NETWORK
TITLE = 1109 - MCC10.3_I811_MA3508 - Zone 1 Burner Fan - Motor

       CALL #"MCC10.3_I811_MA3508"
       (
         CM_No       := 1109 ,
         Unit       :=  ,
         Type       :=  ,
         Tab       := 28 ,
         SubTab       := 3 ,
         Safety       :=  ,
         Disconnect       := LCP131_I811_FN3508_DI_Flt ,
         Protect       := MCC10_I811_FC3508_DI_Flt ,
         RotationFB       :=  ,
         P2002_Current       :=  ,
         P2003_Torque       :=  ,
         P2001_RefVolt       := 460 ,
         EU_Ratio       :=  ,
         Gear_Ratio       :=  ,
         DeAct_Standstill       := T#30s ,
         ID_Free_telegram       :=  ,
         AmpRated       := 3,6 ,
         TorqueRated       :=  ,
         kWRated       := 1.5 ,
         SC_Local       := SL_28_S1 ,
         CM_FRQ        := "dbPlcHmiFRQ".FRQ[1109] ,
       );

NETWORK
TITLE = 1110 - MCC10.3_I521_MA3512 - Zone 2 Disc Filter Cleaning Fan - Motor

       CALL #"MCC10.3_I521_MA3512"
       (
         CM_No       := 1110 ,
         Unit       :=  ,
         Type       :=  ,
         Tab       := 28 ,
         SubTab       := 4 ,
         Safety       :=  ,
         Disconnect       := LCP131_I521_FN3512_DI_Flt ,
         Protect       := MCC10_I521_FC3512_DI_Flt ,
         RotationFB       :=  ,
         P2002_Current       :=  ,
         P2003_Torque       :=  ,
         P2001_RefVolt       := 460 ,
         EU_Ratio       :=  ,
         Gear_Ratio       :=  ,
         DeAct_Standstill       := T#30s ,
         ID_Free_telegram       :=  ,
         AmpRated       := 11 ,
         TorqueRated       :=  ,
         kWRated       := 7.5 ,
         SC_Local       := SL_28_S1 ,
         CM_FRQ        := "dbPlcHmiFRQ".FRQ[1110] ,
       );

NETWORK
TITLE = 1111 - MCC10.2_I621_MA3520 - Zone 2 Circulation Fan  - Motor

       CALL #"MCC10.2_I621_MA3520"
       (
         CM_No       := 1111 ,
         Unit       :=  ,
         Type       :=  ,
         Tab       := 28 ,
         SubTab       := 4 ,
         Safety       :=  ,
         Disconnect       := LCP102_I621_FN3520_DI_Flt ,
         Protect       := MCC10_I621_FC3520_DI_Flt ,
         RotationFB       :=  ,
         P2002_Current       :=  ,
         P2003_Torque       :=  ,
         P2001_RefVolt       := 460 ,
         EU_Ratio       :=  ,
         Gear_Ratio       :=  ,
         DeAct_Standstill       := T#30s ,
         ID_Free_telegram       :=  ,
         AmpRated       := 115 ,
         TorqueRated       :=  ,
         kWRated       := 7.5 ,
         SC_Local       := SL_28_S1 ,
         CM_FRQ        := "dbPlcHmiFRQ".FRQ[1111] ,
       );

NETWORK
TITLE = 1112 - MCC10.3_K911_MA3521 - Dryer 2 Sealing Fan  - Motor

       CALL #"MCC10.3_K911_MA3521"
       (
         CM_No       := 1112 ,
         Unit       :=  ,
         Type       :=  ,
         Tab       := 28 ,
         SubTab       := 1 ,
         Safety       :=  ,
         Disconnect       := LCP131_K911_FN3521_DI_Flt ,
         Protect       := MCC10_K911_FC3521_DI_Flt ,
         RotationFB       :=  ,
         P2002_Current       :=  ,
         P2003_Torque       :=  ,
         P2001_RefVolt       := 460 ,
         EU_Ratio       :=  ,
         Gear_Ratio       :=  ,
         DeAct_Standstill       := T#30s ,
         ID_Free_telegram       :=  ,
         AmpRated       := 5,8 ,
         TorqueRated       :=  ,
         kWRated       := 5.5 ,
         SC_Local       := SL_28_S2 ,
         CM_FRQ        := "dbPlcHmiFRQ".FRQ[1112] ,
       );

NETWORK
TITLE = 1113 - MCC10.3_K511_MA3522 - Zone 3 Disc Filter Cleaning Fan - Motor

       CALL #"MCC10.3_K511_MA3522"
       (
         CM_No       := 1113 ,
         Unit       :=  ,
         Type       :=  ,
         Tab       := 28 ,
         SubTab       := 5 ,
         Safety       :=  ,
         Disconnect       := LCP131_K511_FN3522_DI_Flt ,
         Protect       := MCC10_K511_FC3522_DI_Flt ,
         RotationFB       :=  ,
         P2002_Current       :=  ,
         P2003_Torque       :=  ,
         P2001_RefVolt       := 460 ,
         EU_Ratio       :=  ,
         Gear_Ratio       :=  ,
         DeAct_Standstill       := T#30s ,
         ID_Free_telegram       :=  ,
         AmpRated       := 11 ,
         TorqueRated       :=  ,
         kWRated       := 3 ,
         SC_Local       := SL_28_S2 ,
         CM_FRQ        := "dbPlcHmiFRQ".FRQ[1113] ,
       );

NETWORK
TITLE = 1114 - MCC10.2_K611_MA3530 - Zone 3 Circulation Fan  - Motor

       CALL #"MCC10.2_K611_MA3530"
       (
         CM_No       := 1114 ,
         Unit       :=  ,
         Type       :=  ,
         Tab       := 28 ,
         SubTab       := 5 ,
         Safety       :=  ,
         Disconnect       := LCP103_K611_FN3530_DI_Flt ,
         Protect       := MCC10_K611_FC3530_DI_Flt ,
         RotationFB       :=  ,
         P2002_Current       :=  ,
         P2003_Torque       :=  ,
         P2001_RefVolt       := 460 ,
         EU_Ratio       :=  ,
         Gear_Ratio       :=  ,
         DeAct_Standstill       := T#30s ,
         ID_Free_telegram       :=  ,
         AmpRated       := 115 ,
         TorqueRated       :=  ,
         kWRated       := 3 ,
         SC_Local       := SL_28_S2 ,
         CM_FRQ        := "dbPlcHmiFRQ".FRQ[1114] ,
       );

NETWORK
TITLE = 1115 - MCC10.3_K711_MA3526 - Zone 3 Exhaust Fan - Motor

       CALL #"MCC10.3_K711_MA3526"
       (
         CM_No       := 1115 ,
         Unit       :=  ,
         Type       :=  ,
         Tab       := 28 ,
         SubTab       := 5 ,
         Safety       :=  ,
         Disconnect       := LCP131_K711_FN3526_DI_Flt ,
         Protect       := MCC10_K711_FC3526_DI_Flt ,
         RotationFB       :=  ,
         P2002_Current       :=  ,
         P2003_Torque       :=  ,
         P2001_RefVolt       := 460 ,
         EU_Ratio       :=  ,
         Gear_Ratio       :=  ,
         DeAct_Standstill       := T#30s ,
         ID_Free_telegram       :=  ,
         AmpRated       := 8,6 ,
         TorqueRated       :=  ,
         kWRated       := 1.5 ,
         SC_Local       := SL_28_S2 ,
         CM_FRQ        := "dbPlcHmiFRQ".FRQ[1115] ,
       );

NETWORK
TITLE = 1116 - MCC10.3_K811_MA3528 - Zone 3 Burner Fan - Motor

       CALL #"MCC10.3_K811_MA3528"
       (
         CM_No       := 1116 ,
         Unit       :=  ,
         Type       :=  ,
         Tab       := 28 ,
         SubTab       := 5 ,
         Safety       :=  ,
         Disconnect       := LCP131_K811_FN3528_DI_Flt ,
         Protect       := MCC10_K811_FC3528_DI_Flt ,
         RotationFB       :=  ,
         P2002_Current       :=  ,
         P2003_Torque       :=  ,
         P2001_RefVolt       := 460 ,
         EU_Ratio       :=  ,
         Gear_Ratio       :=  ,
         DeAct_Standstill       := T#30s ,
         ID_Free_telegram       :=  ,
         AmpRated       := 3,6 ,
         TorqueRated       :=  ,
         kWRated       := 7.5 ,
         SC_Local       := SL_28_S2 ,
         CM_FRQ        := "dbPlcHmiFRQ".FRQ[1116] ,
       );

NETWORK
TITLE = 1117 - MCC10.3_K521_MA3532 - Zone 4 Disc Filter Cleaning Fan - Motor

       CALL #"MCC10.3_K521_MA3532"
       (
         CM_No       := 1117 ,
         Unit       :=  ,
         Type       :=  ,
         Tab       := 28 ,
         SubTab       := 6 ,
         Safety       :=  ,
         Disconnect       := LCP131_K521_FN3532_DI_Flt ,
         Protect       := MCC10_K521_FC3532_DI_Flt ,
         RotationFB       :=  ,
         P2002_Current       :=  ,
         P2003_Torque       :=  ,
         P2001_RefVolt       := 460 ,
         EU_Ratio       :=  ,
         Gear_Ratio       :=  ,
         DeAct_Standstill       := T#30s ,
         ID_Free_telegram       :=  ,
         AmpRated       := 11 ,
         TorqueRated       :=  ,
         kWRated       := 7.5 ,
         SC_Local       := SL_28_S2 ,
         CM_FRQ        := "dbPlcHmiFRQ".FRQ[1117] ,
       );

NETWORK
TITLE = 1118 - MCC10.2_K621_MA3540 - Zone 4 Circulation Fan  - Motor

       CALL #"MCC10.2_K621_MA3540"
       (
         CM_No       := 1118 ,
         Unit       :=  ,
         Type       :=  ,
         Tab       := 28 ,
         SubTab       := 6 ,
         Safety       :=  ,
         Disconnect       := LCP104_K621_FN3540_DI_Flt ,
         Protect       := MCC10_K621_FC3540_DI_Flt ,
         RotationFB       :=  ,
         P2002_Current       :=  ,
         P2003_Torque       :=  ,
         P2001_RefVolt       := 460 ,
         EU_Ratio       :=  ,
         Gear_Ratio       :=  ,
         DeAct_Standstill       := T#30s ,
         ID_Free_telegram       :=  ,
         AmpRated       := 115 ,
         TorqueRated       :=  ,
         kWRated       := 5.5 ,
         SC_Local       := SL_28_S2 ,
         CM_FRQ        := "dbPlcHmiFRQ".FRQ[1118] ,
       );

NETWORK
TITLE = 1119 - MCC10.3_K721_MA3536 - Zone 4 Exhaust Fan - Motor

       CALL #"MCC10.3_K721_MA3536"
       (
         CM_No       := 1119 ,
         Unit       :=  ,
         Type       :=  ,
         Tab       := 28 ,
         SubTab       := 6 ,
         Safety       :=  ,
         Disconnect       := LCP131_K721_FN3536_DI_Flt ,
         Protect       := MCC10_K721_FC3536_DI_Flt ,
         RotationFB       :=  ,
         P2002_Current       :=  ,
         P2003_Torque       :=  ,
         P2001_RefVolt       := 460 ,
         EU_Ratio       :=  ,
         Gear_Ratio       :=  ,
         DeAct_Standstill       := T#30s ,
         ID_Free_telegram       :=  ,
         AmpRated       := 8,6 ,
         TorqueRated       :=  ,
         kWRated       := 3 ,
         SC_Local       := SL_28_S2 ,
         CM_FRQ        := "dbPlcHmiFRQ".FRQ[1119] ,
       );

NETWORK
TITLE = 1120 - MCC10.3_K821_MA3538 - Zone 4 Burner Fan - Motor

       CALL #"MCC10.3_K821_MA3538"
       (
         CM_No       := 1120 ,
         Unit       :=  ,
         Type       :=  ,
         Tab       := 28 ,
         SubTab       := 6 ,
         Safety       :=  ,
         Disconnect       := LCP131_K821_FN3538_DI_Flt ,
         Protect       := MCC10_K821_FC3538_DI_Flt ,
         RotationFB       :=  ,
         P2002_Current       :=  ,
         P2003_Torque       :=  ,
         P2001_RefVolt       := 460 ,
         EU_Ratio       :=  ,
         Gear_Ratio       :=  ,
         DeAct_Standstill       := T#30s ,
         ID_Free_telegram       :=  ,
         AmpRated       := 3,6 ,
         TorqueRated       :=  ,
         kWRated       := 3 ,
         SC_Local       := SL_28_S2 ,
         CM_FRQ        := "dbPlcHmiFRQ".FRQ[1120] ,
       );

NETWORK
TITLE = 1121 - MCC11.3_N911_MA3541 - Dryer 3 Sealing Fan  - Motor

       CALL #"MCC11.3_N911_MA3541"
       (
         CM_No       := 1121 ,
         Unit       :=  ,
         Type       :=  ,
         Tab       := 28 ,
         SubTab       := 2 ,
         Safety       :=  ,
         Disconnect       := LCP131_N911_FN3541_DI_Flt ,
         Protect       := MCC11_N911_FC3541_DI_Flt ,
         RotationFB       :=  ,
         P2002_Current       :=  ,
         P2003_Torque       :=  ,
         P2001_RefVolt       := 460 ,
         EU_Ratio       :=  ,
         Gear_Ratio       :=  ,
         DeAct_Standstill       := T#30s ,
         ID_Free_telegram       :=  ,
         AmpRated       := 5,8 ,
         TorqueRated       :=  ,
         kWRated       := 1.5 ,
         SC_Local       := SL_28_S3 ,
         CM_FRQ        := "dbPlcHmiFRQ".FRQ[1121] ,
       );

NETWORK
TITLE = 1122 - MCC11.3_N511_MA3542 - Zone 5 Disc Filter Cleaning Fan - Motor

       CALL #"MCC11.3_N511_MA3542"
       (
         CM_No       := 1122 ,
         Unit       :=  ,
         Type       :=  ,
         Tab       := 28 ,
         SubTab       := 7 ,
         Safety       :=  ,
         Disconnect       := LCP131_N511_FN3542_DI_Flt ,
         Protect       := MCC11_N511_FC3542_DI_Flt ,
         RotationFB       :=  ,
         P2002_Current       :=  ,
         P2003_Torque       :=  ,
         P2001_RefVolt       := 460 ,
         EU_Ratio       :=  ,
         Gear_Ratio       :=  ,
         DeAct_Standstill       := T#30s ,
         ID_Free_telegram       :=  ,
         AmpRated       := 11 ,
         TorqueRated       :=  ,
         kWRated       := 7.5 ,
         SC_Local       := SL_28_S3 ,
         CM_FRQ        := "dbPlcHmiFRQ".FRQ[1122] ,
       );

NETWORK
TITLE = 1123 - MCC11.2_N611_MA3550 - Zone 5 Circulation Fan  - Motor

       CALL #"MCC11.2_N611_MA3550"
       (
         CM_No       := 1123 ,
         Unit       :=  ,
         Type       :=  ,
         Tab       := 28 ,
         SubTab       := 7 ,
         Safety       :=  ,
         Disconnect       := LCP111_N611_FN3550_DI_Flt ,
         Protect       := MCC11_N611_FC3550_DI_Flt ,
         RotationFB       :=  ,
         P2002_Current       :=  ,
         P2003_Torque       :=  ,
         P2001_RefVolt       := 460 ,
         EU_Ratio       :=  ,
         Gear_Ratio       :=  ,
         DeAct_Standstill       := T#30s ,
         ID_Free_telegram       :=  ,
         AmpRated       := 115 ,
         TorqueRated       :=  ,
         kWRated       := 7.5 ,
         SC_Local       := SL_28_S3 ,
         CM_FRQ        := "dbPlcHmiFRQ".FRQ[1123] ,
       );

NETWORK
TITLE = 1124 - MCC11.3_N711_MA3546 - Zone 5 Exhaust Fan - Motor

       CALL #"MCC11.3_N711_MA3546"
       (
         CM_No       := 1124 ,
         Unit       :=  ,
         Type       :=  ,
         Tab       := 28 ,
         SubTab       := 7 ,
         Safety       :=  ,
         Disconnect       := LCP131_N711_FN3546_DI_Flt ,
         Protect       := MCC11_N711_FC3546_DI_Flt ,
         RotationFB       :=  ,
         P2002_Current       :=  ,
         P2003_Torque       :=  ,
         P2001_RefVolt       := 460 ,
         EU_Ratio       :=  ,
         Gear_Ratio       :=  ,
         DeAct_Standstill       := T#30s ,
         ID_Free_telegram       :=  ,
         AmpRated       := 8,6 ,
         TorqueRated       :=  ,
         kWRated       := 5.5 ,
         SC_Local       := SL_28_S3 ,
         CM_FRQ        := "dbPlcHmiFRQ".FRQ[1124] ,
       );

NETWORK
TITLE = 1125 - MCC11.3_N811_MA3548 - Zone 5 Burner Fan - Motor

       CALL #"MCC11.3_N811_MA3548"
       (
         CM_No       := 1125 ,
         Unit       :=  ,
         Type       :=  ,
         Tab       := 28 ,
         SubTab       := 7 ,
         Safety       :=  ,
         Disconnect       := LCP131_N811_FN3548_DI_Flt ,
         Protect       := MCC11_N811_FC3548_DI_Flt ,
         RotationFB       :=  ,
         P2002_Current       :=  ,
         P2003_Torque       :=  ,
         P2001_RefVolt       := 460 ,
         EU_Ratio       :=  ,
         Gear_Ratio       :=  ,
         DeAct_Standstill       := T#30s ,
         ID_Free_telegram       :=  ,
         AmpRated       := 3,6 ,
         TorqueRated       :=  ,
         kWRated       := 3 ,
         SC_Local       := SL_28_S3 ,
         CM_FRQ        := "dbPlcHmiFRQ".FRQ[1125] ,
       );

NETWORK
TITLE = 1126 - MCC11.3_N521_MA3552 - Zone 6 Disc Filter Cleaning Fan - Motor

       CALL #"MCC11.3_N521_MA3552"
       (
         CM_No       := 1126 ,
         Unit       :=  ,
         Type       :=  ,
         Tab       := 28 ,
         SubTab       := 8 ,
         Safety       :=  ,
         Disconnect       := LCP131_N521_FN3552_DI_Flt ,
         Protect       := MCC11_N521_FC3552_DI_Flt ,
         RotationFB       :=  ,
         P2002_Current       :=  ,
         P2003_Torque       :=  ,
         P2001_RefVolt       := 460 ,
         EU_Ratio       :=  ,
         Gear_Ratio       :=  ,
         DeAct_Standstill       := T#30s ,
         ID_Free_telegram       :=  ,
         AmpRated       := 11 ,
         TorqueRated       :=  ,
         kWRated       := 3 ,
         SC_Local       := SL_28_S3 ,
         CM_FRQ        := "dbPlcHmiFRQ".FRQ[1126] ,
       );

NETWORK
TITLE = 1127 - MCC11.2_N621_MA3560 - Zone 6 Circulation Fan  - Motor

       CALL #"MCC11.2_N621_MA3560"
       (
         CM_No       := 1127 ,
         Unit       :=  ,
         Type       :=  ,
         Tab       := 28 ,
         SubTab       := 8 ,
         Safety       :=  ,
         Disconnect       := LCP112_N621_FN3560_DI_Flt ,
         Protect       := MCC11_N621_FC3560_DI_Flt ,
         RotationFB       :=  ,
         P2002_Current       :=  ,
         P2003_Torque       :=  ,
         P2001_RefVolt       := 460 ,
         EU_Ratio       :=  ,
         Gear_Ratio       :=  ,
         DeAct_Standstill       := T#30s ,
         ID_Free_telegram       :=  ,
         AmpRated       := 115 ,
         TorqueRated       :=  ,
         kWRated       := 1.5 ,
         SC_Local       := SL_28_S3 ,
         CM_FRQ        := "dbPlcHmiFRQ".FRQ[1127] ,
       );

NETWORK
TITLE = 1128 - MCC11.3_N721_MA3556 - Zone 6 Exhaust Fan - Motor

       CALL #"MCC11.3_N721_MA3556"
       (
         CM_No       := 1128 ,
         Unit       :=  ,
         Type       :=  ,
         Tab       := 28 ,
         SubTab       := 8 ,
         Safety       :=  ,
         Disconnect       := LCP131_N721_FN3556_DI_Flt ,
         Protect       := MCC11_N721_FC3556_DI_Flt ,
         RotationFB       :=  ,
         P2002_Current       :=  ,
         P2003_Torque       :=  ,
         P2001_RefVolt       := 460 ,
         EU_Ratio       :=  ,
         Gear_Ratio       :=  ,
         DeAct_Standstill       := T#30s ,
         ID_Free_telegram       :=  ,
         AmpRated       := 8,6 ,
         TorqueRated       :=  ,
         kWRated       := 7.5 ,
         SC_Local       := SL_28_S3 ,
         CM_FRQ        := "dbPlcHmiFRQ".FRQ[1128] ,
       );

NETWORK
TITLE = 1129 - MCC11.3_N821_MA3558 - Zone 6 Burner Fan - Motor

       CALL #"MCC11.3_N821_MA3558"
       (
         CM_No       := 1129 ,
         Unit       :=  ,
         Type       :=  ,
         Tab       := 28 ,
         SubTab       := 8 ,
         Safety       :=  ,
         Disconnect       := LCP131_N821_FN3558_DI_Flt ,
         Protect       := MCC11_N821_FC3558_DI_Flt ,
         RotationFB       :=  ,
         P2002_Current       :=  ,
         P2003_Torque       :=  ,
         P2001_RefVolt       := 460 ,
         EU_Ratio       :=  ,
         Gear_Ratio       :=  ,
         DeAct_Standstill       := T#30s ,
         ID_Free_telegram       :=  ,
         AmpRated       := 3,6 ,
         TorqueRated       :=  ,
         kWRated       := 7.5 ,
         SC_Local       := SL_28_S3 ,
         CM_FRQ        := "dbPlcHmiFRQ".FRQ[1129] ,
       );

NETWORK
TITLE = 1130 - MCC11.3_N531_MA3562 - Zone 7 Disc Filter Cleaning Fan - Motor

       CALL #"MCC11.3_N531_MA3562"
       (
         CM_No       := 1130 ,
         Unit       :=  ,
         Type       :=  ,
         Tab       := 28 ,
         SubTab       := 9 ,
         Safety       :=  ,
         Disconnect       := LCP131_N531_FN3562_DI_Flt ,
         Protect       := MCC11_N531_FC3562_DI_Flt ,
         RotationFB       :=  ,
         P2002_Current       :=  ,
         P2003_Torque       :=  ,
         P2001_RefVolt       := 460 ,
         EU_Ratio       :=  ,
         Gear_Ratio       :=  ,
         DeAct_Standstill       := T#30s ,
         ID_Free_telegram       :=  ,
         AmpRated       := 11 ,
         TorqueRated       :=  ,
         kWRated       := 5.5 ,
         SC_Local       := SL_28_S3 ,
         CM_FRQ        := "dbPlcHmiFRQ".FRQ[1130] ,
       );

NETWORK
TITLE = 1131 - MCC11.2_N631_MA3570 - Zone 7 Circulation Fan  - Motor

       CALL #"MCC11.2_N631_MA3570"
       (
         CM_No       := 1131 ,
         Unit       :=  ,
         Type       :=  ,
         Tab       := 28 ,
         SubTab       := 9 ,
         Safety       :=  ,
         Disconnect       := LCP113_N631_FN3570_DI_Flt ,
         Protect       := MCC11_N631_FC3570_DI_Flt ,
         RotationFB       :=  ,
         P2002_Current       :=  ,
         P2003_Torque       :=  ,
         P2001_RefVolt       := 460 ,
         EU_Ratio       :=  ,
         Gear_Ratio       :=  ,
         DeAct_Standstill       := T#30s ,
         ID_Free_telegram       :=  ,
         AmpRated       := 115 ,
         TorqueRated       :=  ,
         kWRated       := 3 ,
         SC_Local       := SL_28_S3 ,
         CM_FRQ        := "dbPlcHmiFRQ".FRQ[1131] ,
       );

NETWORK
TITLE = 1132 - MCC11.3_N731_MA3566 - Zone 7 Exhaust Fan - Motor

       CALL #"MCC11.3_N731_MA3566"
       (
         CM_No       := 1132 ,
         Unit       :=  ,
         Type       :=  ,
         Tab       := 28 ,
         SubTab       := 9 ,
         Safety       :=  ,
         Disconnect       := LCP131_N731_FN3566_DI_Flt ,
         Protect       := MCC11_N731_FC3566_DI_Flt ,
         RotationFB       :=  ,
         P2002_Current       :=  ,
         P2003_Torque       :=  ,
         P2001_RefVolt       := 460 ,
         EU_Ratio       :=  ,
         Gear_Ratio       :=  ,
         DeAct_Standstill       := T#30s ,
         ID_Free_telegram       :=  ,
         AmpRated       := 8,6 ,
         TorqueRated       :=  ,
         kWRated       := 3 ,
         SC_Local       := SL_28_S3 ,
         CM_FRQ        := "dbPlcHmiFRQ".FRQ[1132] ,
       );

NETWORK
TITLE = 1133 - MCC11.3_N831_MA3568 - Zone 7 Burner Fan - Motor

       CALL #"MCC11.3_N831_MA3568"
       (
         CM_No       := 1133 ,
         Unit       :=  ,
         Type       :=  ,
         Tab       := 28 ,
         SubTab       := 9 ,
         Safety       :=  ,
         Disconnect       := LCP131_N831_FN3568_DI_Flt ,
         Protect       := MCC11_N831_FC3568_DI_Flt ,
         RotationFB       :=  ,
         P2002_Current       :=  ,
         P2003_Torque       :=  ,
         P2001_RefVolt       := 460 ,
         EU_Ratio       :=  ,
         Gear_Ratio       :=  ,
         DeAct_Standstill       := T#30s ,
         ID_Free_telegram       :=  ,
         AmpRated       := 3,6 ,
         TorqueRated       :=  ,
         kWRated       := 1.5 ,
         SC_Local       := SL_28_S3 ,
         CM_FRQ        := "dbPlcHmiFRQ".FRQ[1133] ,
       );

NETWORK
TITLE = 1134 - MCC12.1_I311_MA3422 - Dryer 1 Wire Drive Roll - Motor

       CALL #"MCC12.1_I311_MA3422"
       (
         CM_No       := 1134 ,
         Unit       :=  ,
         Type       :=  ,
         Tab       := 3 ,
         SubTab       := 1 ,
         Safety       :=  ,
         Disconnect       := LCP121_I311_FN3422_DI_Flt ,
         Protect       := MCC12_I311_FC3422_DI_Flt ,
         RotationFB       :=  ,
         P2002_Current       :=  ,
         P2003_Torque       :=  ,
         P2001_RefVolt       := 460 ,
         EU_Ratio       :=  ,
         Gear_Ratio       :=  ,
         DeAct_Standstill       := T#30s ,
         ID_Free_telegram       :=  ,
         AmpRated       := 38 ,
         TorqueRated       :=  ,
         kWRated       := 7.5 ,
         SC_Local       := SL_03_S5 ,
         CM_FRQ        := "dbPlcHmiFRQ".FRQ[1134] ,
       );

NETWORK
TITLE = 1135 - MCC12.1_J311_MA3424 - Spray 1 Wire Drive Roll - Motor

       CALL #"MCC12.1_J311_MA3424"
       (
         CM_No       := 1135 ,
         Unit       :=  ,
         Type       :=  ,
         Tab       := 3 ,
         SubTab       := 1 ,
         Safety       :=  ,
         Disconnect       := LCP121_J311_FN3424_DI_Flt ,
         Protect       := MCC12_J311_FC3424_DI_Flt ,
         RotationFB       :=  ,
         P2002_Current       :=  ,
         P2003_Torque       :=  ,
         P2001_RefVolt       := 460 ,
         EU_Ratio       :=  ,
         Gear_Ratio       :=  ,
         DeAct_Standstill       := T#30s ,
         ID_Free_telegram       :=  ,
         AmpRated       := 18,1 ,
         TorqueRated       :=  ,
         kWRated       := 7.5 ,
         SC_Local       := SL_03_S6 ,
         CM_FRQ        := "dbPlcHmiFRQ".FRQ[1135] ,
       );

NETWORK
TITLE = 1136 - MCC12.1_K311_MA3426 - Dryer 2 Wire Drive Roll - Motor

       CALL #"MCC12.1_K311_MA3426"
       (
         CM_No       := 1136 ,
         Unit       :=  ,
         Type       :=  ,
         Tab       := 3 ,
         SubTab       := 1 ,
         Safety       :=  ,
         Disconnect       := LCP122_K311_FN3426_DI_Flt ,
         Protect       := MCC12_K311_FC3426_DI_Flt ,
         RotationFB       :=  ,
         P2002_Current       :=  ,
         P2003_Torque       :=  ,
         P2001_RefVolt       := 460 ,
         EU_Ratio       :=  ,
         Gear_Ratio       :=  ,
         DeAct_Standstill       := T#30s ,
         ID_Free_telegram       :=  ,
         AmpRated       := 38 ,
         TorqueRated       :=  ,
         kWRated       := 5.5 ,
         SC_Local       := SL_03_S7 ,
         CM_FRQ        := "dbPlcHmiFRQ".FRQ[1136] ,
       );

NETWORK
TITLE = 1137 - MCC12.1_L311_MA3428 - Transition Wire Drive Roll - Motor

       CALL #"MCC12.1_L311_MA3428"
       (
         CM_No       := 1137 ,
         Unit       :=  ,
         Type       :=  ,
         Tab       := 3 ,
         SubTab       := 1 ,
         Safety       :=  ,
         Disconnect       := LCP122_L311_FN3428_DI_Flt ,
         Protect       := MCC12_L311_FC3428_DI_Flt ,
         RotationFB       :=  ,
         P2002_Current       :=  ,
         P2003_Torque       :=  ,
         P2001_RefVolt       := 460 ,
         EU_Ratio       :=  ,
         Gear_Ratio       :=  ,
         DeAct_Standstill       := T#30s ,
         ID_Free_telegram       :=  ,
         AmpRated       := 18,1 ,
         TorqueRated       :=  ,
         kWRated       := 3 ,
         SC_Local       := SL_03_S8 ,
         CM_FRQ        := "dbPlcHmiFRQ".FRQ[1137] ,
       );

NETWORK
TITLE = 1138 - MCC12.1_M311_MA3430 - Spray 2 Wire Drive Roll - Motor

       CALL #"MCC12.1_M311_MA3430"
       (
         CM_No       := 1138 ,
         Unit       :=  ,
         Type       :=  ,
         Tab       := 3 ,
         SubTab       := 1 ,
         Safety       :=  ,
         Disconnect       := LCP122_M311_FN3430_DI_Flt ,
         Protect       := MCC12_M311_FC3430_DI_Flt ,
         RotationFB       :=  ,
         P2002_Current       :=  ,
         P2003_Torque       :=  ,
         P2001_RefVolt       := 460 ,
         EU_Ratio       :=  ,
         Gear_Ratio       :=  ,
         DeAct_Standstill       := T#30s ,
         ID_Free_telegram       :=  ,
         AmpRated       := 18,1 ,
         TorqueRated       :=  ,
         kWRated       := 3 ,
         SC_Local       := SL_03_S9 ,
         CM_FRQ        := "dbPlcHmiFRQ".FRQ[1138] ,
       );

NETWORK
TITLE = 1139 - MCC12.2_N311_MA3432 - Dryer 3 Wire Drive Roll - Motor

       CALL #"MCC12.2_N311_MA3432"
       (
         CM_No       := 1139 ,
         Unit       :=  ,
         Type       :=  ,
         Tab       := 3 ,
         SubTab       := 1 ,
         Safety       :=  ,
         Disconnect       := LCP123_N311_FN3432_DI_Flt ,
         Protect       := MCC12_N311_FC3432_DI_Flt ,
         RotationFB       :=  ,
         P2002_Current       :=  ,
         P2003_Torque       :=  ,
         P2001_RefVolt       := 460 ,
         EU_Ratio       :=  ,
         Gear_Ratio       :=  ,
         DeAct_Standstill       := T#30s ,
         ID_Free_telegram       :=  ,
         AmpRated       := 38 ,
         TorqueRated       :=  ,
         kWRated       := 1.5 ,
         SC_Local       := SL_03_S10 ,
         CM_FRQ        := "dbPlcHmiFRQ".FRQ[1139] ,
       );

NETWORK
TITLE = 1140 - MCC12.2_R311_MA3434 - Return Wire 1 Drive Roll - Motor

       CALL #"MCC12.2_R311_MA3434"
       (
         CM_No       := 1140 ,
         Unit       :=  ,
         Type       :=  ,
         Tab       := 3 ,
         SubTab       := 1 ,
         Safety       :=  ,
         Disconnect       := LCP123_R311_FN3434_DI_Flt ,
         Protect       := MCC12_R311_FC3434_DI_Flt ,
         RotationFB       :=  ,
         P2002_Current       :=  ,
         P2003_Torque       :=  ,
         P2001_RefVolt       := 460 ,
         EU_Ratio       :=  ,
         Gear_Ratio       :=  ,
         DeAct_Standstill       := T#30s ,
         ID_Free_telegram       :=  ,
         AmpRated       := 31 ,
         TorqueRated       :=  ,
         kWRated       := 7.5 ,
         SC_Local       := SL_03_S11 ,
         CM_FRQ        := "dbPlcHmiFRQ".FRQ[1140] ,
       );

NETWORK
TITLE = 1141 - MCC12.2_R321_MA3436 - Return Wire 2 Drive Roll - Motor

       CALL #"MCC12.2_R321_MA3436"
       (
         CM_No       := 1141 ,
         Unit       :=  ,
         Type       :=  ,
         Tab       := 3 ,
         SubTab       := 1 ,
         Safety       :=  ,
         Disconnect       := LCP123_R321_FN3436_DI_Flt ,
         Protect       := MCC12_R321_FC3436_DI_Flt ,
         RotationFB       :=  ,
         P2002_Current       :=  ,
         P2003_Torque       :=  ,
         P2001_RefVolt       := 460 ,
         EU_Ratio       :=  ,
         Gear_Ratio       :=  ,
         DeAct_Standstill       := T#30s ,
         ID_Free_telegram       :=  ,
         AmpRated       := 31 ,
         TorqueRated       :=  ,
         kWRated       := 7.5 ,
         SC_Local       := SL_03_S11 ,
         CM_FRQ        := "dbPlcHmiFRQ".FRQ[1141] ,
       );

NETWORK
TITLE = 1142 - MCC12.2_S311_MA3438 - Cooling Wire Drive Roll - Motor

       CALL #"MCC12.2_S311_MA3438"
       (
         CM_No       := 1142 ,
         Unit       :=  ,
         Type       :=  ,
         Tab       := 3 ,
         SubTab       := 1 ,
         Safety       :=  ,
         Disconnect       := LCP122_S311_FN3438_DI_Flt ,
         Protect       := MCC12_S311_FC3438_DI_Flt ,
         RotationFB       :=  ,
         P2002_Current       :=  ,
         P2003_Torque       :=  ,
         P2001_RefVolt       := 460 ,
         EU_Ratio       :=  ,
         Gear_Ratio       :=  ,
         DeAct_Standstill       := T#30s ,
         ID_Free_telegram       :=  ,
         AmpRated       := 18,1 ,
         TorqueRated       :=  ,
         kWRated       := 5.5 ,
         SC_Local       := SL_03_S13 ,
         CM_FRQ        := "dbPlcHmiFRQ".FRQ[1142] ,
       );

NETWORK
TITLE = 1143 - MCC13.3_I211_MA3612 - Dryer 1 Inlet Suction Fan  - Motor

       CALL #"MCC13.3_I211_MA3612"
       (
         CM_No       := 1143 ,
         Unit       :=  ,
         Type       :=  ,
         Tab       := 30 ,
         SubTab       := 4 ,
         Safety       :=  ,
         Disconnect       := LCP131_I211_FN3612_DI_Flt ,
         Protect       := MCC13_I211_FC3612_DI_Flt ,
         RotationFB       :=  ,
         P2002_Current       :=  ,
         P2003_Torque       :=  ,
         P2001_RefVolt       := 460 ,
         EU_Ratio       :=  ,
         Gear_Ratio       :=  ,
         DeAct_Standstill       := T#30s ,
         ID_Free_telegram       :=  ,
         AmpRated       := 8,6 ,
         TorqueRated       :=  ,
         kWRated       := 3 ,
         SC_Local       := SL_30_P ,
         CM_FRQ        := "dbPlcHmiFRQ".FRQ[1143] ,
       );

NETWORK
TITLE = 1144 - MCC13.2_I221_MA3614 - Dryer 1 Outlet Suction Fan  - Motor

       CALL #"MCC13.2_I221_MA3614"
       (
         CM_No       := 1144 ,
         Unit       :=  ,
         Type       :=  ,
         Tab       := 30 ,
         SubTab       := 4 ,
         Safety       :=  ,
         Disconnect       := LCP131_I221_FN3614_DI_Flt ,
         Protect       := MCC13_I221_FC3614_DI_Flt ,
         RotationFB       :=  ,
         P2002_Current       :=  ,
         P2003_Torque       :=  ,
         P2001_RefVolt       := 460 ,
         EU_Ratio       :=  ,
         Gear_Ratio       :=  ,
         DeAct_Standstill       := T#30s ,
         ID_Free_telegram       :=  ,
         AmpRated       := 17,2 ,
         TorqueRated       :=  ,
         kWRated       := 3 ,
         SC_Local       := SL_30_P ,
         CM_FRQ        := "dbPlcHmiFRQ".FRQ[1144] ,
       );

NETWORK
TITLE = 1145 - MCC13.2_I421_MA3616 - Dryer 1 Wire Cleaning Suction Fan - Motor

       CALL #"MCC13.2_I421_MA3616"
       (
         CM_No       := 1145 ,
         Unit       :=  ,
         Type       :=  ,
         Tab       := 30 ,
         SubTab       := 12 ,
         Safety       :=  ,
         Disconnect       := LCP131_I421_FN3616_DI_Flt ,
         Protect       := MCC13_I421_FC3616_DI_Flt ,
         RotationFB       :=  ,
         P2002_Current       :=  ,
         P2003_Torque       :=  ,
         P2001_RefVolt       := 460 ,
         EU_Ratio       :=  ,
         Gear_Ratio       :=  ,
         DeAct_Standstill       := T#30s ,
         ID_Free_telegram       :=  ,
         AmpRated       := 17,2 ,
         TorqueRated       :=  ,
         kWRated       := 1.5 ,
         SC_Local       := SL_30_S5 ,
         CM_FRQ        := "dbPlcHmiFRQ".FRQ[1145] ,
       );

NETWORK
TITLE = 1146 - MCC13.1_I411_MA3618 - Dryer 1 Airknife Fan - Motor

       CALL #"MCC13.1_I411_MA3618"
       (
         CM_No       := 1146 ,
         Unit       :=  ,
         Type       :=  ,
         Tab       := 30 ,
         SubTab       := 12 ,
         Safety       :=  ,
         Disconnect       := LCP131_I411_FN3618_DI_Flt ,
         Protect       := MCC13_I411_FC3618_DI_Flt ,
         RotationFB       :=  ,
         P2002_Current       :=  ,
         P2003_Torque       :=  ,
         P2001_RefVolt       := 460 ,
         EU_Ratio       :=  ,
         Gear_Ratio       :=  ,
         DeAct_Standstill       := T#30s ,
         ID_Free_telegram       :=  ,
         AmpRated       := 28 ,
         TorqueRated       :=  ,
         kWRated       := 7.5 ,
         SC_Local       := SL_30_S5 ,
         CM_FRQ        := "dbPlcHmiFRQ".FRQ[1146] ,
       );

NETWORK
TITLE = 1147 - MCC13.1_K211_MA3620 - Dryer 2 Inlet Suction Fan  - Motor

       CALL #"MCC13.1_K211_MA3620"
       (
         CM_No       := 1147 ,
         Unit       :=  ,
         Type       :=  ,
         Tab       := 30 ,
         SubTab       := 6 ,
         Safety       :=  ,
         Disconnect       := LCP131_K211_FN3620_DI_Flt ,
         Protect       := MCC13_K211_FC3620_DI_Flt ,
         RotationFB       :=  ,
         P2002_Current       :=  ,
         P2003_Torque       :=  ,
         P2001_RefVolt       := 460 ,
         EU_Ratio       :=  ,
         Gear_Ratio       :=  ,
         DeAct_Standstill       := T#30s ,
         ID_Free_telegram       :=  ,
         AmpRated       := 8,6 ,
         TorqueRated       :=  ,
         kWRated       := 7.5 ,
         SC_Local       := SL_30_P ,
         CM_FRQ        := "dbPlcHmiFRQ".FRQ[1147] ,
       );

NETWORK
TITLE = 1148 - MCC13.2_K221_MA3622 - Dryer 2 Outlet Suction Fan  - Motor

       CALL #"MCC13.2_K221_MA3622"
       (
         CM_No       := 1148 ,
         Unit       :=  ,
         Type       :=  ,
         Tab       := 30 ,
         SubTab       := 6 ,
         Safety       :=  ,
         Disconnect       := LCP131_K221_FN3622_DI_Flt ,
         Protect       := MCC13_K221_FC3622_DI_Flt ,
         RotationFB       :=  ,
         P2002_Current       :=  ,
         P2003_Torque       :=  ,
         P2001_RefVolt       := 460 ,
         EU_Ratio       :=  ,
         Gear_Ratio       :=  ,
         DeAct_Standstill       := T#30s ,
         ID_Free_telegram       :=  ,
         AmpRated       := 24 ,
         TorqueRated       :=  ,
         kWRated       := 5.5 ,
         SC_Local       := SL_30_P ,
         CM_FRQ        := "dbPlcHmiFRQ".FRQ[1148] ,
       );

NETWORK
TITLE = 1149 - MCC13.2_K421_MA3624 - Dryer 2 Wire Cleaning Suction Fan - Motor

       CALL #"MCC13.2_K421_MA3624"
       (
         CM_No       := 1149 ,
         Unit       :=  ,
         Type       :=  ,
         Tab       := 30 ,
         SubTab       := 12 ,
         Safety       :=  ,
         Disconnect       := LCP131_K421_FN3624_DI_Flt ,
         Protect       := MCC13_K421_FC3624_DI_Flt ,
         RotationFB       :=  ,
         P2002_Current       :=  ,
         P2003_Torque       :=  ,
         P2001_RefVolt       := 460 ,
         EU_Ratio       :=  ,
         Gear_Ratio       :=  ,
         DeAct_Standstill       := T#30s ,
         ID_Free_telegram       :=  ,
         AmpRated       := 17,2 ,
         TorqueRated       :=  ,
         kWRated       := 3 ,
         SC_Local       := SL_30_S7 ,
         CM_FRQ        := "dbPlcHmiFRQ".FRQ[1149] ,
       );

NETWORK
TITLE = 1150 - MCC13.1_K411_MA3626 - Dryer 2 Airknife Fan - Motor

       CALL #"MCC13.1_K411_MA3626"
       (
         CM_No       := 1150 ,
         Unit       :=  ,
         Type       :=  ,
         Tab       := 30 ,
         SubTab       := 12 ,
         Safety       :=  ,
         Disconnect       := LCP131_K411_FN3626_DI_Flt ,
         Protect       := MCC13_K411_FC3626_DI_Flt ,
         RotationFB       :=  ,
         P2002_Current       :=  ,
         P2003_Torque       :=  ,
         P2001_RefVolt       := 460 ,
         EU_Ratio       :=  ,
         Gear_Ratio       :=  ,
         DeAct_Standstill       := T#30s ,
         ID_Free_telegram       :=  ,
         AmpRated       := 28 ,
         TorqueRated       :=  ,
         kWRated       := 3 ,
         SC_Local       := SL_30_S7 ,
         CM_FRQ        := "dbPlcHmiFRQ".FRQ[1150] ,
       );

NETWORK
TITLE = 1151 - MCC13.3_L211_MA3628 - Transition Wire Fan  - Motor

       CALL #"MCC13.3_L211_MA3628"
       (
         CM_No       := 1151 ,
         Unit       :=  ,
         Type       :=  ,
         Tab       := 30 ,
         SubTab       := 7 ,
         Safety       :=  ,
         Disconnect       := LCP131_L211_FN3628_DI_Flt ,
         Protect       := MCC13_L211_FC3628_DI_Flt ,
         RotationFB       :=  ,
         P2002_Current       :=  ,
         P2003_Torque       :=  ,
         P2001_RefVolt       := 460 ,
         EU_Ratio       :=  ,
         Gear_Ratio       :=  ,
         DeAct_Standstill       := T#30s ,
         ID_Free_telegram       :=  ,
         AmpRated       := 46 ,
         TorqueRated       :=  ,
         kWRated       := 1.5 ,
         SC_Local       := SL_30_P ,
         CM_FRQ        := "dbPlcHmiFRQ".FRQ[1151] ,
       );

NETWORK
TITLE = 1152 - MCC13.1_N221_MA3630 - Dryer 3 Outlet Suction Fan - Motor

       CALL #"MCC13.1_N221_MA3630"
       (
         CM_No       := 1152 ,
         Unit       :=  ,
         Type       :=  ,
         Tab       := 30 ,
         SubTab       := 9 ,
         Safety       :=  ,
         Disconnect       := LCP131_N221_FN3630_DI_Flt ,
         Protect       := MCC13_N221_FC3630_DI_Flt ,
         RotationFB       :=  ,
         P2002_Current       :=  ,
         P2003_Torque       :=  ,
         P2001_RefVolt       := 460 ,
         EU_Ratio       :=  ,
         Gear_Ratio       :=  ,
         DeAct_Standstill       := T#30s ,
         ID_Free_telegram       :=  ,
         AmpRated       := 8,6 ,
         TorqueRated       :=  ,
         kWRated       := 7.5 ,
         SC_Local       := SL_30_P ,
         CM_FRQ        := "dbPlcHmiFRQ".FRQ[1152] ,
       );

NETWORK
TITLE = 1153 - MCC13.2_R211_MA3634 - Return Run 1 Wire Suction Fan 1 - Motor

       CALL #"MCC13.2_R211_MA3634"
       (
         CM_No       := 1153 ,
         Unit       :=  ,
         Type       :=  ,
         Tab       := 30 ,
         SubTab       := 10 ,
         Safety       :=  ,
         Disconnect       := LCP123_R211_FN3634_DI_Flt ,
         Protect       := MCC13_R211_FC3634_DI_Flt ,
         RotationFB       :=  ,
         P2002_Current       :=  ,
         P2003_Torque       :=  ,
         P2001_RefVolt       := 460 ,
         EU_Ratio       :=  ,
         Gear_Ratio       :=  ,
         DeAct_Standstill       := T#30s ,
         ID_Free_telegram       :=  ,
         AmpRated       := 28 ,
         TorqueRated       :=  ,
         kWRated       := 7.5 ,
         SC_Local       := SL_30_P ,
         CM_FRQ        := "dbPlcHmiFRQ".FRQ[1153] ,
       );

NETWORK
TITLE = 1154 - MCC13.2_R212_MA3636 - Return Run 1 Wire Suction Fan 2 - Motor

       CALL #"MCC13.2_R212_MA3636"
       (
         CM_No       := 1154 ,
         Unit       :=  ,
         Type       :=  ,
         Tab       := 30 ,
         SubTab       := 10 ,
         Safety       :=  ,
         Disconnect       := LCP123_R212_FN3636_DI_Flt ,
         Protect       := MCC13_R212_FC3636_DI_Flt ,
         RotationFB       :=  ,
         P2002_Current       :=  ,
         P2003_Torque       :=  ,
         P2001_RefVolt       := 460 ,
         EU_Ratio       :=  ,
         Gear_Ratio       :=  ,
         DeAct_Standstill       := T#30s ,
         ID_Free_telegram       :=  ,
         AmpRated       := 28 ,
         TorqueRated       :=  ,
         kWRated       := 5.5 ,
         SC_Local       := SL_30_P ,
         CM_FRQ        := "dbPlcHmiFRQ".FRQ[1154] ,
       );

NETWORK
TITLE = 1155 - MCC13.2_R221_MA3638 - Return Run 2 Wire Suction Fan 1 - Motor

       CALL #"MCC13.2_R221_MA3638"
       (
         CM_No       := 1155 ,
         Unit       :=  ,
         Type       :=  ,
         Tab       := 30 ,
         SubTab       := 10 ,
         Safety       :=  ,
         Disconnect       := LCP123_R221_FN3638_DI_Flt ,
         Protect       := MCC13_R221_FC3638_DI_Flt ,
         RotationFB       :=  ,
         P2002_Current       :=  ,
         P2003_Torque       :=  ,
         P2001_RefVolt       := 460 ,
         EU_Ratio       :=  ,
         Gear_Ratio       :=  ,
         DeAct_Standstill       := T#30s ,
         ID_Free_telegram       :=  ,
         AmpRated       := 28 ,
         TorqueRated       :=  ,
         kWRated       := 3 ,
         SC_Local       := SL_30_P ,
         CM_FRQ        := "dbPlcHmiFRQ".FRQ[1155] ,
       );

NETWORK
TITLE = 1156 - MCC13.1_R222_MA3640 - Return Run 2 Wire Suction Fan 2 - Motor

       CALL #"MCC13.1_R222_MA3640"
       (
         CM_No       := 1156 ,
         Unit       :=  ,
         Type       :=  ,
         Tab       := 30 ,
         SubTab       := 10 ,
         Safety       :=  ,
         Disconnect       := LCP122_R222_FN3640_DI_Flt ,
         Protect       := MCC13_R222_FC3640_DI_Flt ,
         RotationFB       :=  ,
         P2002_Current       :=  ,
         P2003_Torque       :=  ,
         P2001_RefVolt       := 460 ,
         EU_Ratio       :=  ,
         Gear_Ratio       :=  ,
         DeAct_Standstill       := T#30s ,
         ID_Free_telegram       :=  ,
         AmpRated       := 8,6 ,
         TorqueRated       :=  ,
         kWRated       := 3 ,
         SC_Local       := SL_30_P ,
         CM_FRQ        := "dbPlcHmiFRQ".FRQ[1156] ,
       );

NETWORK
TITLE = 1157 - MCC13.1_R421_MA3642 - Return Run 1 Wire Cleaning Fan - Motor

       CALL #"MCC13.1_R421_MA3642"
       (
         CM_No       := 1157 ,
         Unit       :=  ,
         Type       :=  ,
         Tab       := 30 ,
         SubTab       := 10 ,
         Safety       :=  ,
         Disconnect       := LCP123_R421_FN3642_DI_Flt ,
         Protect       := MCC13_R421_FC3642_DI_Flt ,
         RotationFB       :=  ,
         P2002_Current       :=  ,
         P2003_Torque       :=  ,
         P2001_RefVolt       := 460 ,
         EU_Ratio       :=  ,
         Gear_Ratio       :=  ,
         DeAct_Standstill       := T#30s ,
         ID_Free_telegram       :=  ,
         AmpRated       := 11 ,
         TorqueRated       :=  ,
         kWRated       := 1.5 ,
         SC_Local       := SL_30_S11 ,
         CM_FRQ        := "dbPlcHmiFRQ".FRQ[1157] ,
       );

NETWORK
TITLE = 1158 - MCC13.1_S211_MA3644 - Cooling Section Suction Fan - Motor

       CALL #"MCC13.1_S211_MA3644"
       (
         CM_No       := 1158 ,
         Unit       :=  ,
         Type       :=  ,
         Tab       := 30 ,
         SubTab       := 11 ,
         Safety       :=  ,
         Disconnect       := LCP122_S211_FN3644_DI_Flt ,
         Protect       := MCC13_S211_FC3644_DI_Flt ,
         RotationFB       :=  ,
         P2002_Current       :=  ,
         P2003_Torque       :=  ,
         P2001_RefVolt       := 460 ,
         EU_Ratio       :=  ,
         Gear_Ratio       :=  ,
         DeAct_Standstill       := T#30s ,
         ID_Free_telegram       :=  ,
         AmpRated       := 8,6 ,
         TorqueRated       :=  ,
         kWRated       := 7.5 ,
         SC_Local       := SL_30_P ,
         CM_FRQ        := "dbPlcHmiFRQ".FRQ[1158] ,
       );

NETWORK
TITLE = 1159 - MCC13.3_I111_MA3650 - Münter Box 1 Fan  - Motor

       CALL #"MCC13.3_I111_MA3650"
       (
         CM_No       := 1159 ,
         Unit       :=  ,
         Type       :=  ,
         Tab       := 31 ,
         SubTab       := 1 ,
         Safety       :=  ,
         Disconnect       := LCP131_I111_FN3650_DI_Flt ,
         Protect       := MCC13_I111_FC3650_DI_Flt ,
         RotationFB       :=  ,
         P2002_Current       :=  ,
         P2003_Torque       :=  ,
         P2001_RefVolt       := 480 ,
         EU_Ratio       :=  ,
         Gear_Ratio       :=  ,
         DeAct_Standstill       := T#30s ,
         ID_Free_telegram       :=  ,
         AmpRated       := 48 ,
         TorqueRated       :=  ,
         kWRated       := 7.5 ,
         SC_Local       := SL_30_P ,
         CM_FRQ        := "dbPlcHmiFRQ".FRQ[1159] ,
       );

NETWORK
TITLE = 1160 - MCC13.2_J611_MA3652 - Spray 1 Suction Fan  - Motor

       CALL #"MCC13.2_J611_MA3652"
       (
         CM_No       := 1160 ,
         Unit       :=  ,
         Type       :=  ,
         Tab       := 30 ,
         SubTab       := 5 ,
         Safety       :=  ,
         Disconnect       := LCP131_J611_FN3652_DI_Flt ,
         Protect       := MCC13_J611_FC3652_DI_Flt ,
         RotationFB       :=  ,
         P2002_Current       :=  ,
         P2003_Torque       :=  ,
         P2001_RefVolt       := 480 ,
         EU_Ratio       :=  ,
         Gear_Ratio       :=  ,
         DeAct_Standstill       := T#30s ,
         ID_Free_telegram       :=  ,
         AmpRated       := 23 ,
         TorqueRated       :=  ,
         kWRated       := 5.5 ,
         SC_Local       := SL_30_P ,
         CM_FRQ        := "dbPlcHmiFRQ".FRQ[1160] ,
       );

NETWORK
TITLE = 1161 - MCC13.3_K111_MA3654 - Münter Box 3 Fan  - Motor

       CALL #"MCC13.3_K111_MA3654"
       (
         CM_No       := 1161 ,
         Unit       :=  ,
         Type       :=  ,
         Tab       := 31 ,
         SubTab       := 3 ,
         Safety       :=  ,
         Disconnect       := LCP131_K111_FN3654_DI_Flt ,
         Protect       := MCC13_K111_FC3654_DI_Flt ,
         RotationFB       :=  ,
         P2002_Current       :=  ,
         P2003_Torque       :=  ,
         P2001_RefVolt       := 480 ,
         EU_Ratio       :=  ,
         Gear_Ratio       :=  ,
         DeAct_Standstill       := T#30s ,
         ID_Free_telegram       :=  ,
         AmpRated       := 48 ,
         TorqueRated       :=  ,
         kWRated       := 3 ,
         SC_Local       := SL_30_P ,
         CM_FRQ        := "dbPlcHmiFRQ".FRQ[1161] ,
       );

NETWORK
TITLE = 1162 - MCC13.2_M611_MA3656 - Spray 2 Suction Fan  - Motor

       CALL #"MCC13.2_M611_MA3656"
       (
         CM_No       := 1162 ,
         Unit       :=  ,
         Type       :=  ,
         Tab       := 30 ,
         SubTab       := 8 ,
         Safety       :=  ,
         Disconnect       := LCP131_M611_FN3656_DI_Flt ,
         Protect       := MCC13_M611_FC3656_DI_Flt ,
         RotationFB       :=  ,
         P2002_Current       :=  ,
         P2003_Torque       :=  ,
         P2001_RefVolt       := 480 ,
         EU_Ratio       :=  ,
         Gear_Ratio       :=  ,
         DeAct_Standstill       := T#30s ,
         ID_Free_telegram       :=  ,
         AmpRated       := 23 ,
         TorqueRated       :=  ,
         kWRated       := 3 ,
         SC_Local       := SL_30_P ,
         CM_FRQ        := "dbPlcHmiFRQ".FRQ[1162] ,
       );

NETWORK
TITLE = 1163 - MCC13.3_Q711_MA3662 - Mixing Tank Argitator   - Motor

       CALL #"MCC13.3_Q711_MA3662"
       (
         CM_No       := 1163 ,
         Unit       :=  ,
         Type       :=  ,
         Tab       := 29 ,
         SubTab       := 2 ,
         Safety       :=  ,
         Disconnect       := LCP132_Q711_FN3662_DI_Flt ,
         Protect       := MCC13_Q711_FC3662_DI_Flt ,
         RotationFB       :=  ,
         P2002_Current       :=  ,
         P2003_Torque       :=  ,
         P2001_RefVolt       := 460 ,
         EU_Ratio       :=  ,
         Gear_Ratio       :=  ,
         DeAct_Standstill       := T#30s ,
         ID_Free_telegram       :=  ,
         AmpRated       := 3 ,
         TorqueRated       :=  ,
         kWRated       := 1.5 ,
         SC_Local       := SL_29_P ,
         CM_FRQ        := "dbPlcHmiFRQ".FRQ[1163] ,
       );

NETWORK
TITLE = 1164 - MCC13.3_Q721_MA3664 - Latex Transfer Pump - Motor

       CALL #"MCC13.3_Q721_MA3664"
       (
         CM_No       := 1164 ,
         Unit       :=  ,
         Type       :=  ,
         Tab       := 29 ,
         SubTab       := 2 ,
         Safety       :=  ,
         Disconnect       := LCP132_Q721_FN3664_DI_Flt ,
         Protect       := MCC13_Q721_FC3664_DI_Flt ,
         RotationFB       :=  ,
         P2002_Current       :=  ,
         P2003_Torque       :=  ,
         P2001_RefVolt       := 460 ,
         EU_Ratio       :=  ,
         Gear_Ratio       :=  ,
         DeAct_Standstill       := T#30s ,
         ID_Free_telegram       :=  ,
         AmpRated       := 2,9 ,
         TorqueRated       :=  ,
         kWRated       := 7.5 ,
         SC_Local       := SL_29_P ,
         CM_FRQ        := "dbPlcHmiFRQ".FRQ[1164] ,
       );

NETWORK
TITLE = 1165 - MCC13.3_Q731_MA3666 - Latex Spray 1 - Motor

       CALL #"MCC13.3_Q731_MA3666"
       (
         CM_No       := 1165 ,
         Unit       :=  ,
         Type       :=  ,
         Tab       := 29 ,
         SubTab       := 3 ,
         Safety       :=  ,
         Disconnect       := LCP132_Q731_FN3666_DI_Flt ,
         Protect       := MCC13_Q731_FC3666_DI_Flt ,
         RotationFB       :=  ,
         P2002_Current       :=  ,
         P2003_Torque       :=  ,
         P2001_RefVolt       := 460 ,
         EU_Ratio       :=  ,
         Gear_Ratio       :=  ,
         DeAct_Standstill       := T#30s ,
         ID_Free_telegram       :=  ,
         AmpRated       := 1,5 ,
         TorqueRated       :=  ,
         kWRated       := 7.5 ,
         SC_Local       := SL_29_S1 ,
         CM_FRQ        := "dbPlcHmiFRQ".FRQ[1165] ,
       );

NETWORK
TITLE = 1166 - MCC13.3_Q732_MA3668 - Latex Spray 2 - Motor

       CALL #"MCC13.3_Q732_MA3668"
       (
         CM_No       := 1166 ,
         Unit       :=  ,
         Type       :=  ,
         Tab       := 29 ,
         SubTab       := 4 ,
         Safety       :=  ,
         Disconnect       := LCP132_Q732_FN3668_DI_Flt ,
         Protect       := MCC13_Q732_FC3668_DI_Flt ,
         RotationFB       :=  ,
         P2002_Current       :=  ,
         P2003_Torque       :=  ,
         P2001_RefVolt       := 460 ,
         EU_Ratio       :=  ,
         Gear_Ratio       :=  ,
         DeAct_Standstill       := T#30s ,
         ID_Free_telegram       :=  ,
         AmpRated       := 1,5 ,
         TorqueRated       :=  ,
         kWRated       := 5.5 ,
         SC_Local       := SL_29_S2 ,
         CM_FRQ        := "dbPlcHmiFRQ".FRQ[1166] ,
       );

NETWORK
TITLE = 1167 - MCC13.3_L611_MA3670 - Transition Wire Lift - Motor

       CALL #"MCC13.3_L611_MA3670"
       (
         CM_No       := 1167 ,
         Unit       :=  ,
         Type       :=  ,
         Tab       := 30 ,
         SubTab       := 7 ,
         Safety       :=  ,
         Disconnect       := LCP122_L611_FN3670_DI_Flt ,
         Protect       := MCC13_L611_FC3670_DI_Flt ,
         RotationFB       :=  ,
         P2002_Current       :=  ,
         P2003_Torque       :=  ,
         P2001_RefVolt       := 460 ,
         EU_Ratio       :=  ,
         Gear_Ratio       :=  ,
         DeAct_Standstill       := T#30s ,
         ID_Free_telegram       :=  ,
         AmpRated       := 1,14 ,
         TorqueRated       :=  ,
         kWRated       := 3 ,
         SC_Local       := SL_30_P ,
         CM_FRQ        := "dbPlcHmiFRQ".FRQ[1167] ,
       );

END_FUNCTION_BLOCK
